_CFC_ (* Continuous Function Chart, elements in execution order *)
(* 10s (5s мало) *)
(* 10s (5s мало) *)
#0 TON_AVT:TON(IN: SHU6_V2_YA1_SA7_DI5_A, PT: T#10s)
#1 AND(SHU6_V2_MV2_DI6_RUN, SHU6_P2_YA1_DI1_ZKR)
#2 INT_TO_TIME(ZADER_SHU6_P2_YA1_DI4_OTK)
#3 MUL(#2, 1000)
#4 TON_YA1_Otk:TON(IN: #1, PT: #3)
#5 AND(NOT SHU6_V2_MV2_DI6_RUN, SHU6_P2_YA1_DI2_OTK)
#6 INT_TO_TIME(ZADER_SHU6_P2_YA1_DI3_ZKR)
#7 MUL(#6, 1000)
#8 TON_YA1_ZKR:TON(IN: #5, PT: #7)
#9 AND(SHU6_V2_MV2_DI6_RUN, NOT SHU6_P2_YA1_DI2_OTK)
#10 INT_TO_TIME(ZADER_SHU6_P2_YA1_DI4_OTK)
#11 MUL(#10, 1000)
#12 TON_YA1_N_OTKR:TON(IN: #9, PT: #11)
#13 OR(SHU6_P2_YA1_DI1_ZKR, SHU6_P2_Z_NET_VH_NAPR)
#14 AND(NOT SHU6_V2_MV2_DI6_RUN, NOT #13)
#15 INT_TO_TIME(ZADER_SHU6_P2_YA1_DI3_ZKR)
#16 MUL(#15, 1000)
#17 TON_YA1_N_ZAKR:TON(IN: #14, PT: #16)
#18 OR(#4.Q, #8.Q, #12.Q, #17.Q, YA1_OTKAZ)
#19 AND(#0.Q, #18)
#20 SR_YA1_Otkaz:SR(SET1: #19, RESET: SHU6_P2_SB)
#21 SHU6_P2_Z_YA1_OTKAZ <= #20.Q1
_END_CFC_
(* the same logic as Structured Text *)
(* 10s (5s мало) *)
(* 10s (5s мало) *)
TON_AVT(IN := SHU6_V2_YA1_SA7_DI5_A, PT := T#10s);
TON_YA1_Otk(IN := SHU6_V2_MV2_DI6_RUN AND SHU6_P2_YA1_DI1_ZKR, PT := INT_TO_TIME(ZADER_SHU6_P2_YA1_DI4_OTK) * 1000);
TON_YA1_ZKR(IN := NOT SHU6_V2_MV2_DI6_RUN AND SHU6_P2_YA1_DI2_OTK, PT := INT_TO_TIME(ZADER_SHU6_P2_YA1_DI3_ZKR) * 1000);
TON_YA1_N_OTKR(IN := SHU6_V2_MV2_DI6_RUN AND NOT SHU6_P2_YA1_DI2_OTK, PT := INT_TO_TIME(ZADER_SHU6_P2_YA1_DI4_OTK) * 1000);
TON_YA1_N_ZAKR(IN := NOT SHU6_V2_MV2_DI6_RUN AND NOT (SHU6_P2_YA1_DI1_ZKR OR SHU6_P2_Z_NET_VH_NAPR), PT := INT_TO_TIME(ZADER_SHU6_P2_YA1_DI3_ZKR) * 1000);
SR_YA1_Otkaz(SET1 := TON_AVT.Q AND (TON_YA1_Otk.Q OR TON_YA1_ZKR.Q OR TON_YA1_N_OTKR.Q OR TON_YA1_N_ZAKR.Q OR YA1_OTKAZ), RESET := SHU6_P2_SB);
SHU6_P2_Z_YA1_OTKAZ := SR_YA1_Otkaz.Q1;
END_PROGRAM

(* POU Regim/ALL_Regim, CFC *)
PROGRAM ALL_Regim
VAR
END_VAR
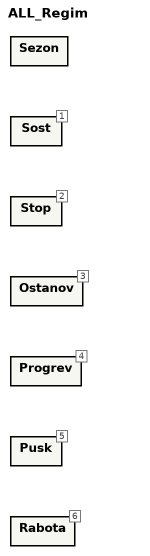
_CFC_ (* Continuous Function Chart, elements in execution order *)
#0 Sezon()
#1 Sost()
#2 Stop()
#3 Ostanov()
#4 Progrev()
#5 Pusk()
#6 Rabota()
_END_CFC_
(* the same logic as Structured Text *)
Sezon();
Sost();
Stop();
Ostanov();
Progrev();
Pusk();
Rabota();
END_PROGRAM

(* POU Regim/Sezon, CFC *)
PROGRAM Sezon
VAR
	RS_Sezon: RS;
	RT_Zima: R_TRIG;
	RT_Leto: R_TRIG;
	RT_Auto: R_TRIG;
	RS_Auto: RS;
	RT_T: R_TRIG;
END_VAR
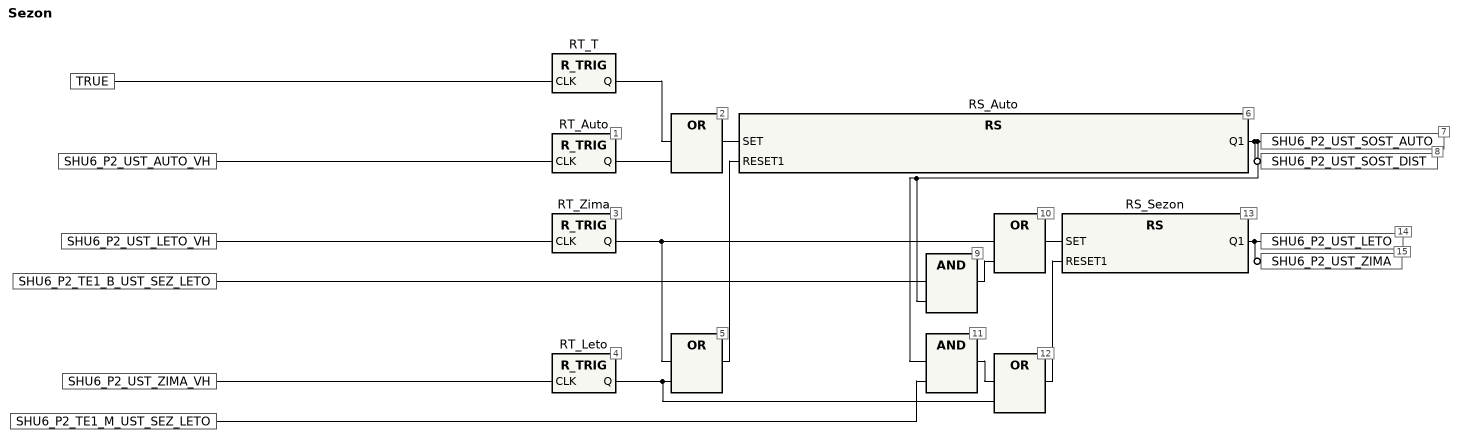
_CFC_ (* Continuous Function Chart, elements in execution order *)
#0 RT_T:R_TRIG(CLK: TRUE)
#1 RT_Auto:R_TRIG(CLK: SHU6_P2_UST_AUTO_VH)
#2 OR(#0.Q, #1.Q)
#3 RT_Zima:R_TRIG(CLK: SHU6_P2_UST_LETO_VH)
#4 RT_Leto:R_TRIG(CLK: SHU6_P2_UST_ZIMA_VH)
#5 OR(#3.Q, #4.Q)
#6 RS_Auto:RS(SET: #2, RESET1: #5)
#7 SHU6_P2_UST_SOST_AUTO <= #6.Q1
#8 SHU6_P2_UST_SOST_DIST <= NOT #6.Q1
#9 AND(SHU6_P2_TE1_B_UST_SEZ_LETO, #6.Q1)
#10 OR(#3.Q, #9)
#11 AND(#6.Q1, SHU6_P2_TE1_M_UST_SEZ_LETO)
#12 OR(#11, #4.Q)
#13 RS_Sezon:RS(SET: #10, RESET1: #12)
#14 SHU6_P2_UST_LETO <= #13.Q1
#15 SHU6_P2_UST_ZIMA <= NOT #13.Q1
_END_CFC_
(* the same logic as Structured Text *)
RT_T(CLK := TRUE);
RT_Auto(CLK := SHU6_P2_UST_AUTO_VH);
RT_Zima(CLK := SHU6_P2_UST_LETO_VH);
RT_Leto(CLK := SHU6_P2_UST_ZIMA_VH);
RS_Auto(SET := RT_T.Q OR RT_Auto.Q, RESET1 := RT_Zima.Q OR RT_Leto.Q);
SHU6_P2_UST_SOST_AUTO := RS_Auto.Q1;
SHU6_P2_UST_SOST_DIST := NOT RS_Auto.Q1;
RS_Sezon(SET := RT_Zima.Q OR (SHU6_P2_TE1_B_UST_SEZ_LETO AND RS_Auto.Q1), RESET1 := (RS_Auto.Q1 AND SHU6_P2_TE1_M_UST_SEZ_LETO) OR RT_Leto.Q);
SHU6_P2_UST_LETO := RS_Sezon.Q1;
SHU6_P2_UST_ZIMA := NOT RS_Sezon.Q1;
END_PROGRAM

(* POU Regim/Sost, CFC *)
PROGRAM Sost
VAR
	RS_Sost: RS;
	RT_PUSK: R_TRIG;
	RT_STOP: R_TRIG;
	RS_Old_Sost: RS;
	TON_Kv1: TON;
	TON_Kv1_1: TON;
	OLD_SOST: BOOL;

	KV1: BOOL;
	RT_PUSK_OLD: R_TRIG;
	CTU_TS: CTU;
	TOF_TS_1: TOF;
	TOF_TS_2: TOF;
	TOF_TS_3: TOF;
	RT_PUSK_OLD1: R_TRIG;
	TON_Kv1_11: TON;
	TON_Kv11: TON;
	TOF_TE_1: TOF;
	TOF_Te_2: TOF;
	TOF_Te_3: TOF;
	CTU_Te: CTU;
END_VAR
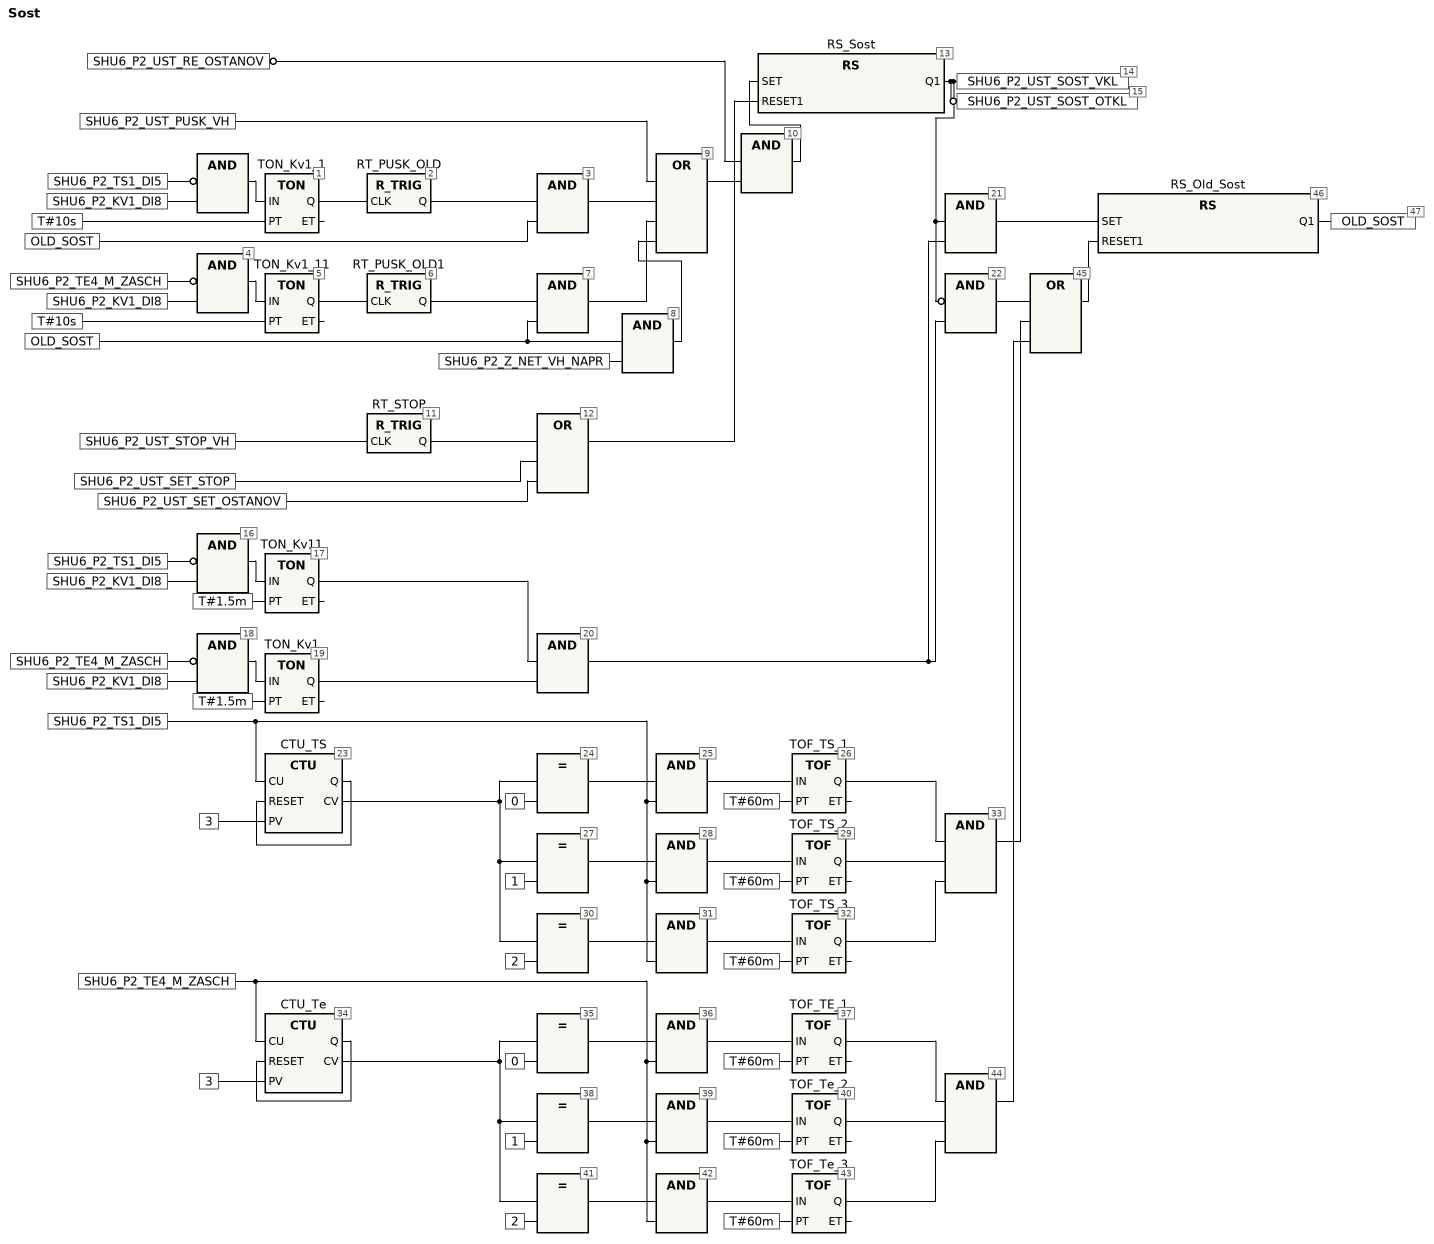
